FUNCTION "LAxisCtrl_UnpubReferencingVelocitySyncAxis" : LReal   // FC30638, SCL
TITLE = LAxisCtrl_UnpubReferencingVelocitySyncAxis
{ S7_Optimized_Access := 'TRUE' }
AUTHOR : tech.team.motioncontrol@siemens.com
FAMILY : AxisCtrl
VERSION : 1.1
// Support: tech.team.motioncontrol@siemens.com
   VAR_INPUT
      axis : TO_SynchronousAxis;   // Axis specification
   END_VAR
   // Ret_Val : axis.Homing.ReferencingVelocity
BEGIN
   // Read axis parameter
   #LAxisCtrl_UnpubReferencingVelocitySyncAxis := #axis.Homing.ReferencingVelocity;
END_FUNCTION

// ===== library: MasterCopy "LAxisCtrl_UnpubSensorTypePosAxis" =====

// folder: LAxisCtrl_Blocks/InternalSubBlocks/SensorType

FUNCTION "LAxisCtrl_UnpubSensorTypePosAxis" : DInt   // FC30643, SCL
TITLE = LAxisCtrl_UnpubSensorTypePosAxis
{ S7_Optimized_Access := 'TRUE' }
AUTHOR : tech.team.motioncontrol@siemens.com
FAMILY : AxisCtrl
VERSION : 1.1
// Support: tech.team.motioncontrol@siemens.com
   VAR_INPUT
      axis : TO_PositioningAxis;   // Axis specification
      index : Int;   // Index of sensor
   END_VAR
   // Ret_Val : axis.Sensor[index].Type
BEGIN
   // Read axis parameter
   #LAxisCtrl_UnpubSensorTypePosAxis := #axis.Sensor[#index].Type;
END_FUNCTION

// ===== library: MasterCopy "LAxisCtrl_UnpubSensorTypeSyncAxis" =====

// folder: LAxisCtrl_Blocks/InternalSubBlocks/SensorType

FUNCTION "LAxisCtrl_UnpubSensorTypeSyncAxis" : DInt   // FC30642, SCL
TITLE = LAxisCtrl_UnpubSensorTypeSyncAxis
{ S7_Optimized_Access := 'TRUE' }
AUTHOR : tech.team.motioncontrol@siemens.com
FAMILY : AxisCtrl
VERSION : 1.1
// Support: tech.team.motioncontrol@siemens.com
   VAR_INPUT
      axis : TO_SynchronousAxis;   // Axis specification
      index : Int;   // Index of sensor
   END_VAR
   // Ret_Val : axis.Sensor[index].Type
BEGIN
   // Read axis parameter
   #LAxisCtrl_UnpubSensorTypeSyncAxis := #axis.Sensor[#index].Type;
END_FUNCTION

// ===== library: MasterCopy "LAxisCtrl_typeGearOutCamOut" =====

// folder: LAxisCtrl_Types/LAxisCtrl_SubTypes

TYPE "LAxisCtrl_typeGearOutCamOut"
TITLE = LAxisCtrl_typeGearOutCamOut
// Support: tech.team.motioncontrol@siemens.com
   STRUCT
      slavePosition : LReal := 0.0;   // Stop position of following axis
      syncProfileReference : DInt := 1;   // Type of desynchronization (0: Desynchronize using dynamic behavior; 1: Desynchronize using leading value distance; 5: Cancel only a pending gearing / camming)
      masterStopDistance : LReal := 0.0;   // Leading value distance when "SyncProfileReference" = 1
      deceleration : LReal := -1.0;   // Deceleration for desynchronization (Value > 0.0: The specified value is used; Value = 0.0: Not permitted; Value < 0.0: Use of the default value configured in the technology object) when "SyncProfileReference" = 0
      jerk : LReal := -1.0;   // Jerk for desynchronization (Value > 0.0: Smooth velocity profile, the specified value is used; Value = 0.0: Trapezoidal velocity profile; Value < 0.0: Use of the default value configured in the technology object) when "SyncProfileReference" = 0
      syncOutDirection : DInt := 3;   // Desynchronization direction (1: Positive direction; 2: Negative direction; 3: Current direction)
      gearOutCamOutMode : DInt := -1;   // -1: Automatic detection whether to use a MC_GearOut or MC_CamOut; 0: Use of MC_GearOut; 1: Use of MC_CamOut
   END_STRUCT;
END_TYPE

// ===== library: MasterCopy "LAxisCtrl_typeGearInRelative" =====

// folder: LAxisCtrl_Types/LAxisCtrl_SubTypes

TYPE "LAxisCtrl_typeGearInRelative"
TITLE = LAxisCtrl_typeGearInRelative
// Support: tech.team.motioncontrol@siemens.com
   STRUCT
      ratioNumerator : DInt := 1;   // Gear ratio numerator (permitted integer values: -2147483648 to 2147483647; value 0 not permitted)
      ratioDenominator : DInt := 1;   // Gear ratio denominator (permitted integer values: 1 to 2147483647)
      acceleration : LReal := -1.0;   // Acceleration for synchronization (Value > 0.0: The specified value is used; Value = 0.0: Not permitted; Value < 0.0: Use of the default value configured in the technology object)
      deceleration : LReal := -1.0;   // Deceleration for synchronization (Value > 0.0: The specified value is used; Value = 0.0: Not permitted; Value < 0.0: Use of the default value configured in the technology object)
      jerk : LReal := -1.0;   // Jerk for synchronization (Value > 0.0: Smooth velocity profile, the specified value is used; Value = 0.0: Trapezoid velocity profile; Value < 0.0: Use of the default value configured in the technology object)
      ratioChangeOnTheFly : Bool := FALSE;   // TRUE: Changing gear ratio on-the-fly; FALSE: Ratio change requires a new rising edge at gearInRelative input
   END_STRUCT;
END_TYPE

// ===== library: MasterCopy "LAxisCtrl_Axis" =====

// folder: LAxisCtrl_Blocks

FUNCTION_BLOCK "LAxisCtrl_Axis"   // FB30616, SCL
TITLE = LAxisCtrl_Axis
{ S7_Optimized_Access := 'TRUE' }
AUTHOR : tech.team.motioncontrol@siemens.com
FAMILY : AxisCtrl
VERSION : 1.2
// Support: tech.team.motioncontrol@siemens.com
   VAR_INPUT
      enable : Bool := FALSE;   // TRUE: Enable functionality of FB
      enableAxis : Bool := FALSE;   // TRUE: Set axis enable; FALSE: Remove axis enable
      resetAxis : Bool := FALSE;   // Rising edge: Acknowledgment of technology alarms or restart of the axis (depending on configuration)
      openBrake : Bool := FALSE;   // TRUE: Unconditionally open holding brake if axis is not enabled (e.g. for service purposes)
      jogForward : Bool := FALSE;   // Rising edge: Move an axis in jog mode (forward); Falling edge: Stop jogging
      jogBackward : Bool := FALSE;   // Rising edge: Move an axis in jog mode (backward); Falling edge: Stop jogging
      moveVelocity : Bool := FALSE;   // Rising edge: Move an axis at constant velocity/speed
      stop : Bool := FALSE;   // Rising edge: Brake an axis until it comes to a standstill. Note: MC_Halt is triggered internally
      fastStop : Bool := FALSE;   // Rising edge: Brake an axis until it comes to a standstill (with fastStop dynamics). Note: MC_Halt is triggered internally
      torqueLimiting : Bool := FALSE;   // TRUE: Enable force/torque limiting
      homing : Bool := FALSE;   // Rising edge: Home axis
      posRelative : Bool := FALSE;   // Rising edge: Move an axis relative to its position when execution of the job began
      posAbsolute : Bool := FALSE;   // Rising edge: Move an axis to an absolute position
      posSuperimposed : Bool := FALSE;   // Rising edge: Start a superimposed positioning
      gearInRelative : Bool := FALSE;   // Rising edge: Start a gearing operation (relative)
      gearInAbsolute : Bool := FALSE;   // Rising edge: Start a gearing operation (absolute)
      gearOutCamOut : Bool := FALSE;   // Rising edge: End a gearing/camming operation
      camIn : Bool := FALSE;   // Rising edge: Start a camming operation
      phasing : Bool := FALSE;   // Rising edge: Start a phasing operation
      offset : Bool := FALSE;   // Rising edge: Start an offset operation
      axis : DB_ANY := 0;   // Reference to axis technology object to be controlled
      master : DB_ANY := 0;   // Reference to leading axis technology object for synchronous motion
      cam : DB_ANY := 0;   // Cam technology object
      configuration : "LAxisCtrl_typeAxisConfig";   // Structure for parameters
   END_VAR
   VAR_OUTPUT
      valid : Bool := FALSE;   // TRUE: Valid set of output values available at the FB
      busy : Bool := FALSE;   // TRUE: FB is working and new output values can be expected
      error : Bool := FALSE;   // TRUE: An error occurred while processing the FB
      status : Word := 16#7000;   // Current status of FB (16#0000 - 16#7FFF: Status of the FB, 16#8000 - 16#FFFF: Error identification)
      statusText : String[#STATUS_TEXT_LENGTH] := STRING#'STATUS_NO_CALL';   // Text of current status of FB
      subfunctionStatus : Word;   // Status of internally called subfunctions (ErrorID of Motion Control instructions)
      axisEnabled : Bool := FALSE;   // TRUE: The technology object is enabled. Motion commands can be executed
      resetActive : Bool := FALSE;   // TRUE: Reset/Restart of the axis is active
      commandBusy : Bool := FALSE;   // TRUE: The selected basic motion command is being executed
      commandDone : Bool := FALSE;   // TRUE: The selected basic motion command has completed without error
      commandAborted : Bool := FALSE;   // TRUE: The selected basic motion command has been aborted
      inVelocity : Bool := FALSE;   // TRUE: The setpoint velocity/speed was reached and will be maintained
      inLimitation : Bool := FALSE;   // TRUE: The drive is operating at the force/torque limit
      homingCommandBusy : Bool := FALSE;   // TRUE: Homing command is being executed
      homingCommandDone : Bool := FALSE;   // TRUE: Homing command has completed without error
      homingCommandAborted : Bool := FALSE;   // TRUE: Homing command has been aborted
      superimposedBusy : Bool := FALSE;   // TRUE: The selected superimposed motion command is being executed
      superimposedDone : Bool := FALSE;   // TRUE: The selected superimposed motion command has completed without error
      superimposedAborted : Bool := FALSE;   // TRUE: The selected superimposed motion command has been aborted
      superimposedStart : Bool := FALSE;   // TRUE: The selected superimposed motion is active
      inClamping : Bool := FALSE;   // TRUE: The drive is kept at the fixed stop (clamping), the axis position is within the positioning tolerance
      startSync : Bool := FALSE;   // TRUE: The axis is synchronizing to the leading axis / desynchronizing from the leading axis
      inSync : Bool := FALSE;   // TRUE: The axis is synchronized to the leading axis
      endOfProfile : Bool := FALSE;   // TRUE: The end of the cam has been reached. The output is displayed for at least one call when the cam is used cyclically
      inSimulation : Bool := FALSE;   // TRUE: Synchronous operation is being simulated
      jogSelected : Bool := FALSE;   // TRUE: Jogging is active
      moveVelocitySelected : Bool := FALSE;   // TRUE: Moving with constant velocity/speed is active
      stopSelected : Bool := FALSE;   // TRUE: Stopping is active
      fastStopSelected : Bool := FALSE;   // TRUE: Stopping is active (with fastStop dynamics)
      torqueLimitingSelected : Bool := FALSE;   // TRUE: Force/Torque limiting is active
      homingSelected : Bool := FALSE;   // TRUE: Homing is active
      posRelativeSelected : Bool := FALSE;   // TRUE: Relative positioning is active
      posAbsoluteSelected : Bool := FALSE;   // TRUE: Absolute positioning is active
      posSuperimposedSelected : Bool := FALSE;   // TRUE: Superimposed positioning is active (See also outputs: superimposedBusy, superimposedDone, superimposedAborted)
      gearInRelativeSelected : Bool := FALSE;   // TRUE: Relative gearing is active (See also outputs: commandBusy, commandDone, commandAborted, inSync)
      gearInAbsoluteSelected : Bool := FALSE;   // TRUE: Absolute gearing is active (See also outputs: commandBusy, commandDone, commandAborted, startSync, inSync)
      gearOutCamOutSelected : Bool := FALSE;   // TRUE: End a gearing/camming operation is active (See also outputs: commandBusy, commandDone, commandAborted, startSync)
      camInSelected : Bool := FALSE;   // TRUE: Camming is active (See also outputs: commandBusy, commandDone, commandAborted, startSync, inSync)
      phasingSelected : Bool := FALSE;   // TRUE: Phasing is active (See also outputs: superimposedBusy, superimposedDone, superimposedAborted, superimposedStart)
      offsetSelected : Bool := FALSE;   // TRUE: Offset is active (See also outputs: superimposedBusy, superimposedDone, superimposedAborted, superimposedStart)
      diagnostics : "LAxisCtrl_typeDiagnostics";   // Diagnostics structure
   END_VAR
   VAR
      statStatusOld : Word;   // Old value of statStatus
      statStatusText : String[#STATUS_TEXT_LENGTH] := STRING#'STATUS_NO_CALL';   // Internal text of current status of FB
      statErrorUserCleared : Bool := FALSE;   // Error occurred that can only be solved by user; rising edge at enable input necessary
      statErrorAutoCleared : Bool := FALSE;   // Error occurred that can be acknowledged by FB
      statStatus : Word := 16#7000;   // Internal variable for status
      statSubfunctionStatus : Word := 16#0000;   // Internal variable for subfunction status
      statDiagnostics : "LAxisCtrl_typeDiagnostics";   // Internal variable for diagnostics
      statEnableOld : Bool := FALSE;   // Old value of enable for edge detection
      statFBState : SInt := 1;   // State of FB (function block state machine)
      statFirstCycleReset : Bool := TRUE;   // TRUE: First cycle of reset command
      statPowerErrorOld : Bool := FALSE;   // Old value of LAnyAxis_MC_Power.error
      statResetState : Int := 0;   // State of reset command
      statFirstCycleResetError : Bool := FALSE;   // TRUE: First cycle of error in reset command
      statExtendedCommand : DWord := 16#0000_0000;   // Variable for requested extended command (e.g. resetAxis, torquelimiting, homing)
      statExtendedCommandOld : DWord := 16#0000_0000;   // Old value of variable for requested extended command
      statEnableAxisOld : Bool := FALSE;   // Old value of enableAxis for edge detection
      statEmptyDiagnostics : "LAxisCtrl_typeDiagnostics";   // Internal empty diagnostic structure
      statHomingOld : Bool := FALSE;   // Old value of variable for homing command input
      statFirstCycleHoming : Bool := TRUE;   // TRUE: First cycle in homing command
      statPassiveHomingState : DInt := -10;   // Current selected passive homing mode
      statExeOfHoming : Int := 1;   // Current state of execution of homing command
      statBasicCommand : DWord := 16#0000_0000;   // Variable for requested basic motion command
      statBasicCommandOld : DWord := 16#0000_0000;   // Old value of variable for requested basic motion command
      statBasicMotionState : DInt := 0;   // State of selected basic motion command
      statExeOfBasicMotion : Int := 1;   // State of execution of current state of basic motion
      statFirstCycleBasicMotion : Bool := TRUE;   // TRUE: First cycle in respective state fo basic motion functionality
      statApplicativeBasicMotionError : Bool := FALSE;   // TRUE: applicative error occurred (e.g. invalid direction configured)
      statVelocityChangeOnTheFly : Bool := FALSE;   // Velocity change on the fly is active
      statBasicVelocity : LReal := 0.0;   // Internal variable for velocity
      statBasicAcceleration : LReal := 0.0;   // Internal variable for acceleration
      statBasicAbortAcceleration : Bool := FALSE;   // FALSE: The current acceleration at the start of the job is reduced using the configured jerk. Afterwards, the deceleration builds up; TRUE: The acceleration is set to 0.0 at the start of the job, and the deceleration immediately builds up.
      statBasicDeceleration : LReal := 0.0;   // Internal variable for deceleration
      statBasicJerk : LReal := 0.0;   // Internal variable for jerk
      statPositionControlled : Bool := TRUE;   // FALSE: Non position-controlled operation; TRUE: Position-controlled operation
      statFirstCycleDone : Bool := FALSE;   // TRUE: First cycle of done at fastStop
      statTorqueLimitingState : SInt := 0;   // Current executed state for torquelimiting functionality
      statTorqueLimitingErrorOld : Bool := FALSE;   // TRUE: Error at Torquelimiting occurred last cycle
      statTorqueLimit : LReal := -1.0;   // Value of force/torque limiting (in the configured unit of measurement)
      statJogMode : DInt := 0;   // Current selected jog mode
      statDirection : Int := 0;   // Internal variable for direction of rotation of the axis
      statStopWithoutSignalization : Bool;   // Internal variable for stopOnError function
      statBrakeOpened : Bool;   // Brake is openend
      statBrakeChangeActive : Bool;   // Brake change active
      statOpenBrakeOld : Bool;   // Edge detection
      statSupImpVelocity : LReal := 0.0;   // Internal variable for velocity
      statSupImpAcceleration : LReal := 0.0;   // Internal variable for acceleration
      statSupImpDeceleration : LReal := 0.0;   // Internal variable for deceleration
      statSupImpJerk : LReal := 0.0;   // Internal variable for jerk
      statHomingPosition : LReal := 0.0;   // The specified value is used according to the selected "Mode".
      statHomingSubState : SInt := 0;   // Current subState of execution of homing functionality
      statIncJogSubState : SInt := 0;   // Current subState of execution of jog incremental functionality
      statIncJogStartPosition : LReal := 0.0;   // Last stored axis position (for incremental jogging)
      statIncJogDirectionOld : Int := 0;   // Old value of direction of executing incremental jogging
      statIncrement : LReal := 0.0;   // Jog Incremental: distance of Increment (positive or negative)
      statIncJogDistance : LReal := 0.0;   // Jog Incremental: current distance to destination position
      statResetIncJog : Bool := TRUE;   // TRUE: First cycle in incremental jogging state (detection of new increment)
      statPosition : LReal := 0.0;   // Internal variable for position
      statPositionChangeOnTheFly : Bool := FALSE;   // Position change on the fly is active
      statHomingMode : Int := 0;   // Operating Mode of LAnyAxis_MC_HOME command
      statActiveHomingState : DInt := -10;   // Current selected active homing mode
      statSupImpCommand : DWord := 16#0000_0000;   // Variable for requested superimposed motion command
      statSupImpCommandOld : DWord := 16#0000_0000;   // Old value of variable for requested superimposed motion command
      statSupImpMotionState : DInt := 0;   // Current selected superimposed motion functionality
      statExeOfSupImpMotionState : Int := 1;   // Current state of execution of superimposed basic motion
      statFirstCycleSupImpMotion : Bool := TRUE;   // TRUE: First cycle in positioning (superimposed) functionality
      statSupImpMotionPosition : LReal := 0.0;   // Position setpoint (for posSuperimposed command)
      statApplicativeSupImpMotionError : Bool := FALSE;   // TRUE: applicative error occurred (e.g. invalid direction configured)
      statRatioChangeOnTheFly : Bool := FALSE;   // Ratio change on the fly is active
      statRatioNumerator : DInt := 1;   // Gear ratio numerator
      statRatioDenominator : DInt := 1;   // Gear ratio denominator
      statChangePhaseShiftOnTheFly : Bool := FALSE;   // Phase shift change on the fly is active
      statChangeOffsetOnTheFly : Bool := FALSE;   // Offset change on the fly is active
      statPhaseShift : LReal := 0.0;   // Relative/Absolute master value shift
      statPhaseAbsolute : Bool := TRUE;   // Indicates the type of phase shift (TRUE: The phase shift is taken over as an absolute value; FALSE: The phase shift is added to an existing offset)
      statOffsetAbsolute : Bool := FALSE;   // Indicates the type of offset shift (TRUE: The offset shift is taken over as an absolute value; FALSE: The offset shift is added to an existing offset)
      statOffsetValue : LReal := 0.0;   // Relative/Absolute offset
      statTypeAxis : Int;   // Type of axis
      statSupImpProfileReference : DInt := 0;   // Internal variable
      statSupImpDistance : LReal := 0.0;   // Internal variable
      statSupImpStartPosition : LReal := 0.0;   // Internal variable
      statSupImpDirection : DInt := 0;   // Internal variable
      statEnableAxis : Bool := FALSE;   // Internal variable for enabling axis
      statSyncMotionSimulationState : SInt := 0;   // Current executed state for synchronized motion simulation
      statSynchronizedMotionErrorOld : Bool := FALSE;   // Old value of LAnyAxis_MC_SynchronizedMotionSimulation.error
      statMainSelectionState : Int := 0;   // Current executed State for execution of basic motion commands or reset of waiting gearing / camming commands
      statMasterSyncPosition : LReal := 0.0;   // Synchronous position of leading axis. Position of the following axis starting from which the leading and following axes move synchronously
      statSlaveSyncPosition : LReal := 0.0;   // Synchronous position of leading axis. Position of the leading axis starting from which the leading and following axes move synchronously
      statBasicSyncDirection : DInt := 1;   // Direction of synchronization
      statBasicMasterStartDistance : LReal := 0.0;   // Master value distance (when "SyncProfileReference" = 1)
      statBasicSyncProfileReference : DInt := 0;   // Type of synchronization
      statApplicationMode : DInt := 0;   // Application of cam
      statCam : DB_ANY := 0;   // Internal variable for cam
      statWaitingFunctionState : DInt := 0;   // Internal variable for waiting function state
      statWaitingFunctionStateAbortAutomatic : DInt := -1;   // Internal variable for waiting function state
      statFunctionState : DInt := 0;   // Internal variable for function state
      statGearAndCamOutMode : DInt := 0;   // Internal variable
      statSyncOutState : DInt;   // Internal variable
      statAxis : DB_ANY;   // Internal axis reference
      instPower : "LAnyAxis_MC_Power";   // Instance of LAnyAxis_MC_Power
      instReset : "LAnyAxis_MC_Reset";   // Instance of LAnyAxis_MC_Reset
      instHome : "LAnyAxis_MC_Home";   // Instance of LAnyAxis_MC_Home
      instHalt : "LAnyAxis_MC_Halt";   // Instance of LAnyAxis_MC_Halt
      instMoveJog : "LAnyAxis_MC_MoveJog";   // Instance of LAnyAxis_MC_MoveJog
      instTorqueLimiting : "LAnyAxis_MC_TorqueLimiting";   // Instance of LAnyAxis_MC_TorqueLimiting
      instMoveVelocity : "LAnyAxis_MC_MoveVelocity";   // Instance of LAnyAxis_MC_MoveVelocity
      instSetAxisSTW : "LAnyAxis_MC_SetAxisSTW";   // Instance of LAnyAxis_MC_SetAxisSTW
      instMoveRelative : "LAnyAxis_MC_MoveRelative";   // Instance of LAnyAxis_MC_MoveRelative
      instMoveAbsolute : "LAnyAxis_MC_MoveAbsolute";   // Instance of LAnyAxis_MC_MoveAbsolute
      instMoveSuperimposed : "LAnyAxis_MC_MoveSuperimposed";   // Instance of LAnyAxis_MC_MoveSuperimposed
      instGearIn : "LAnyAxis_MC_GearIn";   // Instance of LAnyAxis_MC_GearIn
      instPhasingAbsolute : "LAnyAxis_MC_PhasingAbsolute";   // Instance of LAnyAxis_MC_PhasingAbsolute
      instPhasingRelative : "LAnyAxis_MC_PhasingRelative";   // Instance of LAnyAxis_MC_PhasingRelative
      instOffsetAbsolute : "LAnyAxis_MC_OffsetAbsolute";   // Instance of LAnyAxis_MC_OffsetAbsolute
      instOffsetRelative : "LAnyAxis_MC_OffsetRelative";   // Instance of LAnyAxis_MC_OffsetRelative
      instGearInPos : "LAnyAxis_MC_GearInPos";   // Instance of LAnyAxis_MC_GearInPos
      instGearOut : "LAnyAxis_MC_GearOut";   // Instance of LAnyAxis_MC_GearOut
      instCamIn : "LAnyAxis_MC_CamIn";   // Instance of MC_CamIn
      instCamOut : "LAnyAxis_MC_CamOut";   // Instance of LAnyAxis_MC_CamOut
      instSyncMotionSimulation : "LAnyAxis_MC_SynchronizedMotionSimulation";   // Instance of LAnyAxis_MC_SynchronizedMotionSimulation
   END_VAR
   VAR_TEMP
      tempEnable : Bool;   // Temporary variable for enable FB
      tempNewExtendedCmd : DInt;   // Temporary variable for extended command
      tempEnableAxis : Bool;   // Temporary variable for enableAxis
      tempErrorInCmd : Bool;   // Temporary variable for error in actual command
      tempRisingCmd : DWord;   // Temporary DWord which indicates all rising edges of command word
      tempStopCmdSelected : Bool;   // TRUE: Stop or faststop selected in current cycle
      tempOpenBrake : Bool;   // Temporary variable for open brake
      tempDword : DWord;   // Temporary DWord for evaluation of rising edges of basic command word
      tempIndex : Int;   // Temporary index
      tempCountRisEdges : USInt;   // Temporary counter for rising edges in command word
      tempNewBasicMotionCmd : DInt;   // Temporary variable for basic motion command
      tempStateChangeActive : Bool;   // TRUE: State change is active, stay in loop for one more cycle
      tempStatusWord : DWord;   // Temporary variable for statusword of axis
      tempNewSupImpCmd : DInt;   // Temporary variable for superimposed motion command
      tempHoming : Bool;   // Temporary variable for homing command
   END_VAR
   VAR CONSTANT
      EXTERNAL_ENCODER : Int := 1;   // Axis type: External encoder
      SPEED_AXIS : Int := 2;   // Axis type: Speed axis
      POS_AXIS : Int := 3;   // Axis type: Positioning axis
      SYNC_AXIS : Int := 4;   // Axis type: Synchronous axis
      STATUS_TEXT_LENGTH : Int := 39;   // Length of status text
      AXIS_MOTION : SInt := 1;   // State of FB: MotionState, new commands are evaluated
      FB_ERROR : SInt := 5;   // State of FB: Error, falling edge at FB_ENABLE required
      CMD_NO_SELECTION : DWord := 16#0000_0000;   // No command is selected
      NO_SELECTION : Int := 0;   // State of basicMotion/superimposedMotion: No execution of a command
      AXIS_FAST_STOPPING : SInt := 2;   // State of FB: StoppingState, MC_HALT is executed, new commands are not evaluated
      AXIS_STOP_ON_ERROR_SELECTION : SInt := 3;   // State of FB: ErrorState: Selection if StopOnError must be executed (depending on configuration)
      AXIS_STOP_ON_ERROR_EXECUTION : SInt := 4;   // State of FB: ErrorState: Execution of StopOnError
      FAST_STOP_SELECTED : Int := 1;   // State of basicMotion: Execution of fast stop command
      STOP_SELECTED : Int := 2;   // State of basicMotion: Execution of stop command
      JOG_FORWARD_SELECTED : Int := 4;   // State of basicMotion: Execution of jog forward command
      JOG_BACKWARD_SELECTED : Int := 8;   // State of basicMotion: Execution of jog backward command
      JOG_FW_AND_BW_SELECTED : Int := 12;   // State of basicMotion: Execution of jog command if forward and backward are selected
      MOVE_VELOCITY_SELECTED : Int := 16;   // State of basicMotion: Execution of move velocity command
      ACTIVE_HOMING_SELECTED : Int := 1024;   // State of basicMotion: Execution of active homing command
      POS_RELATIVE_SELECTED : Int := 32;   // State of basicMotion: Execution of position command (relative)
      POS_ABSOLUTE_SELECTED : Int := 64;   // State of basicMotion: Execution of position command (absolute)
      GEAR_IN_RELATIVE_SELECTED : Int := 128;   // State of basicMotion: Execution of gearIn command
      GEAR_IN_ABSOLUTE_SELECTED : Int := 256;   // State of basicMotion: Execution of gearInPos command
      CAM_IN_SELECTED : Int := 512;   // State of basicMotion: Execution of camIn command
      GEAR_OUT_CAM_OUT_SELECTED : Int := 2048;   // State of basicMotion: Execution of gear and camOut command
      POS_SUPERIMPOSED_SELECTED : Int := 1;   // State of superimposedMotion: Execution of posSuperimposed command
      PHASING_SELECTED : Int := 2;   // State of superimposedMotion: Execution of phasing command
      OFFSET_SELECTED : Int := 4;   // State of superimposedMotion: Execution of offset command
      CMD_IDLE : Int := 0;   // State of basicMotion command: No execution
      CMD_BUSY : Int := 1;   // State of basicMotion command: Subsequent call
      CMD_DONE : Int := 2;   // State of basicMotion command: Finished with "DONE"
      CMD_ABORTED : Int := 4;   // State of basicMotion command: Finished with "ABORTED"
      CMD_ERROR : Int := 8;   // State of basicMotion command: Finished with "ERROR"
      CMD_END_PROCESS : Int := 16;   // State of basicMotion command: Finished with other reason
      JOG_MODE_CONTINUOUS : Int := 0;   // Jogmode continuous selected (MC_MOVEJOG)
      NO_TORQUE_LIMITING_ACTIVE : SInt := 0;   // State of torquelimiting command: Not enabled
      TORQUE_LIMTING_SELECTED : SInt := 1;   // State of torquelimiting command: Torquelimiting is active
      TORQUE_LIMITING_DISABLE : SInt := 10;   // State of torquelimiting command: Torquelimiting is disabling
      BITPOSITION_BASIC_MOTION_CMD : SInt := 4;   // First bitposition for detecting rising edges at basic motion command word
      BIT_POS_LAST : SInt := 15;   // Last bitposition for detecting rising edges at command word
      SPECIFIED_DIR : Int := 0;   // The sign of the velocity specified at the "Velocity" parameter defines the direction of rotation.
      MASK_STW_BIT12 : Word := 16#1000;   // Bit 12 in STW
      NO_HOMING_ACTIVE : SInt := -10;   // State of homing command: No homing active
      STANDARD_HOMING : SInt := -1;   // State of homing command: (Standard) homing with MC_HOME
      BITPOSITION_SUPERIMPOSED_MOTION_CMD : SInt := 0;   // First bitposition for detecting rising edges at superimposed motion command word
      FIXED_STOP_DETECTION_ACTIVE : SInt := 2;   // State of torquelimiting command: Homing on fixed stop is active
      FIXED_STOP_DETECTION_FINISHED : SInt := 3;   // State of torquelimiting command: Homing on fixed stop is finished
      FIXED_STOP_DETECTION_ERROR_IN_CLAMPING : SInt := 5;   // State of torquelimiting command: Error occurred at homing on fixed stop process, axis is in clamping
      FIXED_STOP_DETECTION_ERROR_NOT_IN_CLAMPING : SInt := 6;   // State of torquelimiting command: Error occurred at homing on fixed stop process, axis is not in clamping
      HOMING_ON_FIXED_STOP : SInt := 0;   // State of homing command: Applicative homing on fixed stop process active
      HOMING_ON_FIXED_STOP_WITH_MOVING_OUT_OF_CLAMPING : SInt := 1;   // State of homing command: Applicative homing on fixed stop with moving out of clamping process active.
      HOMING_ON_FIXED_STOP_WITH_MOVING_TO_TARGET_POSITION : SInt := 2;   // State of homing command: Applicative homing on fixed stop with moving to target position process active.
      DISTANCE_SCALING : LReal := 1.05;   // Scaling factor for moving out of clamping. 1.0 = positioning window
      MODE_FIXED_STOP_DETECTION : Int := 1;   // Fixed stop detection (Mode for MC_TORQUELIMITING)
      FORWARD_DIR : Int := 1;   // Positive/Forward direction of rotation
      BACKWARD_DIR : Int := 2;   // Negative/Backward direction of rotation
      SHORTEST_WAY_DIR : Int := 3;   // Shortest path
      DIRECT_HOMING : Int := 0;   // Direct homing (absolute). Parameter "position" at MC_HOME is effective
      ACTIVE_HOMING : Int := 3;   // Active homing. Parameter "position" at MC_HOME is effective
      ACTIVE_HOMING_TO_DEF_VALUE : Int := 5;   // Active homing. The configured home position value in technology object is effective
      ABSOLUTE_ENCODER_ADJUSTMENT : Int := 7;   // Absolute encoder adjustment (absolute)
      INCREMENTAL_ENCODER : Int := 0;   // Encodertype INCREMENTAL
      HOMING_IDLE : SInt := 0;   // SubState of homing on fixed stop process: Idle
      HOMING_FIXED_STOP_DETECTION : SInt := 1;   // SubState of homing on fixed stop process: Detecting fixed stop
      HOMING_PROCESS : SInt := 2;   // SubState of homing on fixed stop process: Homeprocess (MC_HOME)
      HOMING_POSITION : SInt := 3;   // SubState of homing on fixed stop process: Positioning to homeposition
      INC_JOG_IDLE : SInt := 0;   // Substate of incremental jog process: Idle
      INC_JOG_START : SInt := 1;   // Substate of incremental jog process: Start moving
      INC_JOG_STOP : SInt := 3;   // Substate of incremental jog process: Stop moving
      JOG_MODE_NEW_INCREMENT : Int := 1;   // Jogmode incremental selected - start always with new increment when command is selected
      JOG_MODE_CONTINUE_INCREMENT : Int := 2;   // Jogmode incremental selected - continue with increment when command is selected again
      APPLICATION_MODE_ONCE : Int := 0;   // Application of the cam: Once/not cyclic (MC_CAMIN)
      CALL_BASIC_MOTION : Int := 0;   // State of MainSelectionState: Regular execution of basic motion commands
      ABORT_WAITING_GEARINPOS_OR_CAMIN : Int := 1;   // State of MainSelectionState: Reset of waiting synchronous commands
      AXIS_NOT_IN_SIM : SInt := 0;   // State of motionSimulation: Axis is not in simulation
      AXIS_STATE_SET_SIM : SInt := 1;   // State of motionSimulation: Setting axis in simulation
      AXIS_DISABLE : SInt := 2;   // State of motionSimulation: Disable axis
      AXIS_STATE_IN_SIM : SInt := 3;   // State of motionSimulation: Axis is in simulation
      AXIS_ENABLE : SInt := 4;   // State of motionSimulation: Enable axis
      AXIS_STATE_RESET_SIM : SInt := 5;   // State of motionSimulation: Resetting axis simulation
      CANCEL_ONLY_WAITING_GEARING_CAMMING : DInt := 5;   // Mode for MC_GearOut / MC_CamOut instruction
      WFS_FS_NO_OPERATION : DInt;   // No operation active or waiting
      WFS_FS_GEARIN : DInt := 1;   // Function state / Waiting function state: GearIn
      WFS_FS_GEARINPOS : DInt := 2;   // Function state / Waiting function state: GearInPos
      WFS_FS_CAMIN : DInt := 3;   // Function state / Waiting function state: CamIn
      WFS_FS_GEAROUT : DInt := 4;   // Function state / Waiting function state: Gearout
      WFS_FS_CAMOUT : DInt := 5;   // Function state / Waiting function state: CamOut
      SYNCOUT_MODE_AUTOMATIC : DInt := -1;   // GearOutCamOut mode: Automatic
      SYNCOUT_MODE_GEAROUT : DInt := 0;   // GearOutCamOut mode: GearOut
      SYNCOUT_MODE_CAMOUT : DInt := 1;   // GearOutCamOut mode: CamOut
      SYNCOUT_STATE_CHECK_WAITING : Int := 1;   // Sync out state
      SYNCOUT_STATE_GEAROUT_WAITING_BUSY : Int := 2;   // Sync out state
      SYNCOUT_STATE_CAMOUT_WAITING_BUSY : Int := 3;   // Sync out state
      SYNCOUT_STATE_CHECK_ACTIVE : Int := 4;   // Sync out state
      SYNCOUT_STATE_GEAROUT_ACTIVE_BUSY : Int := 5;   // Sync out state
      SYNCOUT_STATE_CAMOUT_ACTIVE_BUSY : Int := 6;   // Sync out state
      SYNCOUT_STATE_DONE : Int := 7;   // Sync out state
      SYNCOUT_STATE_ABORTED : Int := 8;   // Sync out state
      SYNCOUT_STATE_ERROR : Int := 9;   // Sync out state
      STATUS_NO_CALL : Word := 16#7000;   // No call of FB
      STATUS_FB_FIRST_CALL : Word := 16#7001;   // First cycle of FB after enabling
      STATUS_SUBSEQUENT_CALL : Word := 16#7002;   // FB enabled
      ERR_INVALID_BASIC_MOTION_CMD : Word := 16#8001;   // Invalid basic command selected (rising edge at 2 or more basic motion command inputs)
      ERR_INVALID_EXTENDED_CMD : Word := 16#8002;   // Invalid extended command selected (rising edge at torque limiting and homing on fixed stop)
      ERR_INVALID_SUPERIMPOSED_MOTION_CMD : Word := 16#8003;   // Invalid superimposed command selected (rising edge at 2 or more superimposed motion command inputs)
      ERR_INVALID_GEAROUT_CAMOUT_MODE : Word := 16#820D;   // Error invalid mode for gearOutCamOut instruction
      ERR_INVALID_SYNCHRONIZED_EXTENDED_MODE : Word := 16#820E;   // Error invalid extended mode for synchronized motion simulation functionality
      ERR_INVALID_JOG_MODE : Word := 16#8201;   // Invalid jog mode selected
      ERR_INVALID_HOMING_EXTENDED_MODE : Word := 16#8202;   // Command Error: Invalid extended homing mode selected
      ERR_TORQUE_LIMITING_NOT_ALLOWED : Word := 16#8203;   // Error during extended homing command - torque limiting not allowed during homing on fixed stop is active or axis in clamping
      ERR_INVALID_JOG_DIR : Word := 16#8204;   // Invalid direction selected (jog forward and jog backward)
      ERR_INVALID_POS_RELATIVE_DIR : Word := 16#8205;   // Invalid direction is set for relative positioning command
      ERR_INVALID_POS_SUPERIMPOSED_DIR : Word := 16#8206;   // Invalid direction is set for superimposed positioning command
      ERR_HOMING_MODE_NOT_ALLOWED : Word := 16#8207;   // Passive/Direct homing is not allowed during extended homing mode (homing on fixed stop process) is active
      ERR_MODULO_NOT_ALLOWED : Word := 16#8208;   // Extended homing mode (homing on fixed stop process) is not allowed with modulo axis
      ERR_INVALID_TORQUE_LIMIT : Word := 16#8209;   // Configured torque limit value for extended homing mode (homing on fixed stop process) = 0
      ERR_INVALID_VELOCITY : Word := 16#820A;   // Configured velocity (in technology object) for active homing = 0
      ERR_INVALID_AXIS : Word := 16#820B;   // Illegal specification of the technology object
      ERR_INVALID_TARGET_POSITION : Word := 16#820C;   // Invalid target position configured for extended homing mode
      ERR_MC_POWER : Word := 16#8600;   // Error occurred during MC_POWER command
      ERR_MC_RESET : Word := 16#8601;   // Error occurred during MC_RESET command
      ERR_MC_HOME : Word := 16#8602;   // Error occurred during MC_HOME command
      ERR_MC_TORQUELIMITING : Word := 16#8603;   // Error occurred during MC_TORQUELIMITING command
      ERR_MC_HALT : Word := 16#8604;   // Error occurred during MC_HALT command
      ERR_MC_MOVEJOG : Word := 16#8605;   // Error occurred during MC_MOVEJOG command (continuous jogging)
      ERR_MC_MOVEVELOCITY : Word := 16#8606;   // Error occurred during MC_MOVEVELOCITY command
      ERR_MC_MOVERELATIVE : Word := 16#8607;   // Error occurred during MC_MOVERELATIVE command
      ERR_MC_MOVEABSOLUTE : Word := 16#8608;   // Error occurred during MC_MOVEABSOLUTE command
      ERR_MC_MOVESUPERIMPOSED : Word := 16#8609;   // Error occurred during MC_MOVESUPERIMPOSED command
      ERR_MC_GEARIN : Word := 16#860A;   // Error occurred during MC_GEARIN command
      ERR_MC_PHASINGABSOLUTE : Word := 16#860B;   // Error occurred during MC_PHASINGABSOLUTE command
      ERR_MC_PHASINGRELATIVE : Word := 16#860C;   // Error occurred during MC_PHASINGRELATIVE command
      ERR_MC_CAMIN : Word := 16#860D;   // Error occurred during MC_CAMIN command
      ERR_MC_GEARINPOS : Word := 16#860E;   // Error occurred during MC_GEARINPOS command
      ERR_MC_SYNCHRONIZEDMOTIONSIMULATION : Word := 16#860F;   // Error occurred during MC_SYNCHRONIZEDMOTIONSIMULATION command
      ERR_MC_OFFSETABSOLUTE : Word := 16#8610;   // Error occurred during MC_OFFSETABSOLUTE command
      ERR_MC_OFFSETRELATIVE : Word := 16#8611;   // Error occurred during MC_OFFSETRELATIVE command
      ERR_MC_CAMOUT : Word := 16#8612;   // Error occurred during MC_CAMOUT command
      ERR_MC_GEAROUT : Word := 16#8613;   // Error occurred during MC_GEAROUT command
      ERR_UNDEFINED_FB_STATE : Word := 16#8700;   // Error due to an undefined FB state
      ERR_UNDEFINED_RESET_STATE : Word := 16#8701;   // Error due to an undefined reset state
      ERR_UNDEFINED_BASIC_MOTION_STATE : Word := 16#8702;   // Error due to an undefined basic motion state
      ERR_UNDEFINED_TORQUE_LIMITING_STATE : Word := 16#8703;   // Error due to an undefined torque limiting state
      ERR_UNDEFINED_INCREMENTAL_JOG_STATE : Word := 16#8704;   // Error due to an undefined incremental jog state
      ERR_UNDEFINED_INCREMENTAL_JOG_SUBSTATE : Word := 16#8705;   // Error due to an undefined incremental jog substate
      ERR_UNDEFINED_EXTENDED_HOMING_STATE : Word := 16#8706;   // Error due to an undefined homing state
      ERR_UNDEFINED_EXTENDED_HOMING_SUBSTATE : Word := 16#8707;   // Error due to an undefined homing substate
      ERR_UNDEFINED_SUPERIMPOSED_MOTION_STATE : Word := 16#8708;   // Error due to an undefined superimposed motion state
      ERR_UNDEFINED_MOTION_SIMULATION_STATE : Word := 16#8709;   // Error due to an undefined synchronized motion simulation state
      ERR_UNDEFINED_MAIN_SELECTION_STATE : Word := 16#870A;   // Error due to an undefined main selection state
   END_VAR
BEGIN
   REGION HEADER
     //================================================================================
     // SIEMENS AG
     // (c)Copyright 2021 All Rights Reserved
     //--------------------------------------------------------------------------------
     // Library: LAxisCtrl 
     // Tested with: S7-1515T-2 PN
     // Engineering: TIA Portal V17
     // Restrictions: -
     // Requirements: S7-1500/S7-1500T FW 2.9
     //               LAnyAxis V1.1                                                                                         
     // Functionality: This function block offers basic functionalities for axis control
     // Support: tech.team.motioncontrol@siemens.com
     // Note: Parameter comments are only available in language 'English (United States)'
     //--------------------------------------------------------------------------------
     // Change log table:
     // Version  Date        Expert in charge  Changes applied
     // 01.00.01 12.10.2016  RS                First released version
     // 01.00.02 29.03.2017  RS                Added support information
     //                                        TorqueLimiting at FB Enable                                                   
     //                                        Block is compilable with V14 SP1
     //                                        Output 'done' is set at endOfProfile of CamIn command (applicationMode ONCE)  
     //                                        fastStop: Use TO emergency stop deceleration in case of configured value <= 0 
     //                                        fastStop: Configured jerk value is always used                                
     // 01.00.03 14.06.2017  RS                Reset MC_TORQUELIMITING instance with disable of FB                           
     //                                        Bugfix of error handling for MC_TORQUELIMITING                                
     //                                        Homing on fixed stop: Use always torque value in homing configuration         
     // 01.00.04 14.12.2017  RS                Initialize diagnostics at rising edge of torquelimiting command               
     //                                        Check of cam (with TYPEOFDB) at start of camIn command                        
     // 01.00.05 30.09.2019  RS                Bugfixes
     //                                        Dont abort waiting sync commands if new gearinAbsolute or camIn or gearIn commands are set   
     //                                        Ratio on the fly: use also new dynamics if "on the fly value" changed         
     //                                        Stop on Error function: No error display if error at MC_Halt                  
     //                                        New extended homing mode: 1: Homing on fixed stop with moving out of clamping                        
     // 01.01.00 31.03.2020  RS                New output "subfunctionStatus"
     //                                        Change of parameter configuration: INOUT --> IN
     //                                        New input: "open brake"                                                       
     //                                        Optimized function: "abort waiting gearing commands"                          
     //                                        Stop on Error function: Error and status outputs remain also if internally        
     //                                        called MC_Halt instruction is executed                                        
     //                                        Output "diagnostics" is only written at end of block                          
     // 01.02.00 26.04.2021  RS                New output "statusText"
     //                                        New extended homing mode: 2: Homing on fixed stop with moving to target position   
     //                                        New feature: Automatic enabling of synchronized motion simulation when axis gets disabled  
     //                                        Update Motion Control V6.0 (MC_Offset_XXX, MC_Phasing_XXX, MC_GearOut; MC_CamOut)         
     //                                        FastStop command aborts waiting synchronous operations                        
     //                                        Bugfix synchronized motion simulation
     // 01.02.01 01.10.2021  RS                Bugfix synchronized motion simulation ('syncMotionSimulationExtendedMode' = -1):
     //                                        Axis is disabled (powered off) now, when parameter 'syncMotionSimulation' is set
     //                                        and no synchronous operation is active (<TO>.StatusWord.X22 = TRUE)
     //================================================================================
   END_REGION

   //----------------------------------------------------------------------------------------------
   // Enable / disable FB
   //----------------------------------------------------------------------------------------------
   REGION ENABLE_FB
     #tempEnable := #enable; // Create temporary process image
     IF NOT #tempEnable AND #statEnableOld THEN
       REGION FALLING_EDGE_AT_ENABLE_FB

         // Reset outputs 
         // ==========================================================
         // Error and valid outputs are reset with falling edge of enable input
         #error := FALSE;
         #valid := FALSE;
         #status := #STATUS_NO_CALL;
         #statusText := STRING#'STATUS_NO_CALL';
         #subfunctionStatus := #statSubfunctionStatus := 16#0; // V1.1.0

         // Reset status outputs
         #axisEnabled := FALSE;
         #resetActive := FALSE;

         // Reset outputs for homing commands
         #homingCommandBusy := FALSE;
         #homingCommandDone := FALSE;
         #homingCommandAborted := FALSE;
         #homingSelected := FALSE;
         // Reset outputs for torquelimiting command
         #torqueLimitingSelected := FALSE;
         #inLimitation := FALSE;

         // Reset outputs for basic motion commands
         #commandDone := FALSE;
         #commandBusy := FALSE;
         #commandAborted := FALSE;
         #inVelocity := FALSE;
         #fastStopSelected := FALSE;
         #stopSelected := FALSE;
         #jogSelected := FALSE;
         #moveVelocitySelected := FALSE;
         // Outputs for for up to LAxisCtrl_PosAxis
         #posRelativeSelected := FALSE;
         #posAbsoluteSelected := FALSE;
         #inClamping := FALSE;

         // Reset outputs for superimposed motion commands
         #superimposedBusy := FALSE;
         #superimposedDone := FALSE;
         #superimposedAborted := FALSE;
         #superimposedStart := FALSE;
         #posSuperimposedSelected := FALSE;
         #startSync := FALSE;
         #inSync := FALSE;
         #endOfProfile := FALSE;
         #gearInRelativeSelected := FALSE;
         #inSimulation := FALSE;
         #gearInAbsoluteSelected := FALSE;
         #phasingSelected := FALSE;
         #offsetSelected := FALSE;
         #camInSelected := FALSE;
         #gearOutCamOutSelected := FALSE;

         // Reset internal variables
         // ==========================================================
         #statErrorUserCleared := FALSE;
         #statErrorAutoCleared := FALSE;
         #statStatus := #STATUS_NO_CALL;
         #statStatusOld := 16#0000;
         #statDiagnostics := #statEmptyDiagnostics;

         #statFBState := #AXIS_MOTION;
         #statFirstCycleReset := FALSE;
         #statPowerErrorOld := FALSE;
         #statResetState := #CMD_IDLE;
         #statFirstCycleResetError := FALSE;

         #statExtendedCommand := #CMD_NO_SELECTION;
         #statExtendedCommandOld := #CMD_NO_SELECTION;
         #statEnableAxisOld := FALSE;
         #statHomingOld := FALSE;
         #statFirstCycleHoming := FALSE;
         #statPassiveHomingState := #NO_HOMING_ACTIVE;
         #statExeOfHoming := #CMD_BUSY;
         #statBasicCommand := #CMD_NO_SELECTION;
         #statBasicCommandOld := #CMD_NO_SELECTION;
         #statBasicMotionState := #NO_SELECTION;
         #statExeOfBasicMotion := #CMD_BUSY;
         #statFirstCycleBasicMotion := FALSE;
         #statApplicativeBasicMotionError := FALSE;
         #statVelocityChangeOnTheFly := FALSE;
         #statBasicVelocity := 0.0;
         #statBasicAcceleration := 0.0;
         #statBasicAbortAcceleration := FALSE;
         #statBasicDeceleration := 0.0;
         #statBasicJerk := 0.0;

         #statPositionControlled := TRUE;
         #statFirstCycleDone := FALSE;

         #statTorqueLimitingState := #NO_TORQUE_LIMITING_ACTIVE;
         #statTorqueLimitingErrorOld := FALSE;
         #statTorqueLimit := -1.0;
         #statJogMode := #JOG_MODE_CONTINUOUS;
         #statDirection := #SPECIFIED_DIR;

         #statSupImpVelocity := 0.0;
         #statSupImpAcceleration := 0.0;
         #statSupImpDeceleration := 0.0;
         #statSupImpJerk := 0.0;

         #statHomingPosition := 0.0;
         #statHomingSubState := #HOMING_IDLE;
         #statIncJogSubState := #INC_JOG_IDLE;
         #statIncJogStartPosition := 0.0;
         #statIncJogDirectionOld := 0;
         #statIncrement := 0.0;
         #statIncJogDistance := 0.0;
         #statResetIncJog := TRUE;
         #statPosition := 0.0;
         #statPositionChangeOnTheFly := FALSE;

         #statHomingMode := #DIRECT_HOMING;
         #statActiveHomingState := #NO_HOMING_ACTIVE;
         #statSupImpCommand := #CMD_NO_SELECTION;
         #statSupImpCommandOld := #CMD_NO_SELECTION;
         #statSupImpMotionState := #NO_SELECTION;
         #statExeOfSupImpMotionState := #CMD_BUSY;
         #statFirstCycleSupImpMotion := FALSE;
         #statSupImpMotionPosition := 0.0;
         #statApplicativeSupImpMotionError := FALSE;
         #statRatioChangeOnTheFly := FALSE;
         #statRatioNumerator := 0;
         #statRatioDenominator := 0;
         // Tags for synchronized motion simulation
         #statChangePhaseShiftOnTheFly := FALSE;
         #statChangeOffsetOnTheFly := FALSE;
         #statPhaseShift := 0.0;
         #statOffsetValue := 0.0;
         #statPhaseAbsolute := TRUE;
         #statOffsetAbsolute := TRUE;
         #statEnableAxis := FALSE;
         #statSyncMotionSimulationState := #AXIS_NOT_IN_SIM;
         #statSynchronizedMotionErrorOld := FALSE;
         #statMainSelectionState := 0;
         #statMasterSyncPosition := 0.0;
         #statSlaveSyncPosition := 0.0;
         #statBasicSyncDirection := #FORWARD_DIR;
         #statBasicMasterStartDistance := 0.0;
         #statBasicSyncProfileReference := 0;
         #statApplicationMode := 0;

         #statSupImpProfileReference := 0;
         #statSupImpDistance := 0.0;
         #statSupImpStartPosition := 0.0;
         #statSupImpDirection := 0;
         #statWaitingFunctionState := 0;
         #statWaitingFunctionStateAbortAutomatic := -1;
         #statFunctionState := 0;
         // ===========================================================

         // Disable Axis
         IF (#instPower.Busy = TRUE) THEN
           #instPower(Axis := #statAxis,
                      Enable := FALSE,
                      StartMode := #configuration.power.startMode,
                      StopMode := #configuration.power.stopMode);
           // Check if error occurred
           IF (#instPower.Error = TRUE) THEN
             // Write only diagnostics if error occurred at falling edge of MC_POWER
             #diagnostics.status := #ERR_MC_POWER;
             #diagnostics.subfunctionStatus := #instPower.ErrorID;
             #diagnostics.basicMotionState := #statBasicMotionState;
             #diagnostics.superimposedMotionState := #statSupImpMotionState;
           END_IF;
         END_IF;

         // Set old value of enable for edge detection and end execution
         #statEnableOld := #tempEnable;
         RETURN;
       END_REGION

       // Check if FB is enabled - first cycle
     ELSIF #tempEnable AND NOT #statEnableOld THEN
       REGION FB_RISING_EDGE_AT_ENABLE_FB
         // Busy is set at rising edge of enable input
         #busy := TRUE;
         #status := #STATUS_FB_FIRST_CALL;
         #statusText := STRING#'STATUS_FB_FIRST_CALL';
         // StatStatus will be written in next cycle
         #statStatus := #STATUS_SUBSEQUENT_CALL;
         #statStatusText := STRING#'STATUS_SUBSEQUENT_CALL';

         // Reset error and diagnostics outputs
         #statErrorUserCleared := FALSE;
         #statErrorAutoCleared := FALSE;
         #diagnostics := #statEmptyDiagnostics;
         #statDiagnostics := #statEmptyDiagnostics;

         // Copy inputs
         #statExtendedCommand.%X0 := #resetAxis;
         #statBasicCommand.%X8 := #gearInAbsolute;
         #statBasicCommand.%X9 := #camIn;
         #statBasicCommand.%X11 := #gearOutCamOut;
         #statSupImpCommand.%X1 := #phasing;
         #statSupImpCommand.%X2 := #offset;
         #statBasicCommand.%X7 := #gearInRelative;
         #statBasicCommand.%X5 := #posRelative;
         #statBasicCommand.%X6 := #posAbsolute;
         #statSupImpCommand.%X0 := #posSuperimposed;
         #statSupImpCommandOld := #statSupImpCommand;
         // #statExtendedCommand.%X1 := #torqueLimiting;  // V1.0.2 Removed for activation at FB Enable 

         #statBasicCommand.%X0 := #fastStop;
         #statBasicCommand.%X1 := #stop;
         #statBasicCommand.%X2 := #jogForward;
         #statBasicCommand.%X3 := #jogBackward;
         #statBasicCommand.%X4 := #moveVelocity;
         #statBasicCommandOld := #statBasicCommand;
         // Set old value of homing input
         #statHomingOld := #homing;

         #statExtendedCommandOld := #statExtendedCommand;
         // Set old value of enable for edge detection and end execution
         #statEnableOld := #tempEnable;

         CASE TypeOfDB(#axis) OF
           TO_SYNCHRONOUSAXIS:
             #statTypeAxis := #SYNC_AXIS;
             #statAxis := #axis;

           TO_POSITIONINGAXIS:
             #statTypeAxis := #POS_AXIS;
             #statAxis := #axis;

           TO_SPEEDAXIS:
             #statTypeAxis := #SPEED_AXIS;
             #statAxis := #axis;

           TO_EXTERNALENCODER:
             // Valid axis
             #statAxis := #axis;
             #statTypeAxis := #EXTERNAL_ENCODER;

           ELSE
             // Invalid axis
             #error := TRUE;
             #statErrorUserCleared := TRUE;
             #status := #ERR_INVALID_AXIS;
             #statusText := STRING#'ERR_INVALID_AXIS';
             #diagnostics.status := #ERR_INVALID_AXIS;
         END_CASE;
         RETURN;
       END_REGION

       // Check if function block is disabled or UserClearedError is present
     ELSIF NOT #tempEnable OR #statErrorUserCleared THEN
       REGION FB_DISABLED
         IF (#tempEnable = FALSE) THEN
           #status := #STATUS_NO_CALL;
           #statusText := STRING#'STATUS_NO_CALL';
         END_IF;

         // Disable Axis
         IF (#instPower.Busy = TRUE) THEN
           #instPower(Axis := #statAxis,
                      Enable := FALSE,
                      StartMode := #configuration.power.startMode,
                      StopMode := #configuration.power.stopMode);
           // Check if error occurred
           IF (#instPower.Error = TRUE) THEN
             #diagnostics.status := #ERR_MC_POWER;
             #diagnostics.subfunctionStatus := #instPower.ErrorID;
             #diagnostics.basicMotionState := #statBasicMotionState;
             #diagnostics.superimposedMotionState := #statSupImpMotionState;
           END_IF;
         ELSE
           // V1.00.03 Reset if torque limiting is busy and axis is disabled 
           IF (#instTorqueLimiting.Busy = TRUE)
             OR (#instSyncMotionSimulation.Busy = TRUE)
           THEN
             #instTorqueLimiting(Axis := #statAxis,
                                 Enable := FALSE);
             // V1.2.0 Disable synchronized motion simulation 
             #instSyncMotionSimulation(Slave := #axis,
                                       Enable := FALSE);
           ELSE
             #busy := FALSE;
           END_IF;
         END_IF;

         #statEnableOld := #tempEnable;
         RETURN;
       END_REGION

     ELSE
       REGION FB_ENABLED
         // Copy extended inputs
         #statExtendedCommand.%X0 := #resetAxis;
         #tempEnableAxis := #enableAxis;
         #statExtendedCommand.%X1 := #torqueLimiting;
         #statBasicCommand.%X0 := #fastStop;
         #statBasicCommand.%X1 := #stop;
         #statBasicCommand.%X2 := #jogForward;
         #statBasicCommand.%X3 := #jogBackward;
         #statBasicCommand.%X4 := #moveVelocity;
         #tempOpenBrake := #openBrake;
         #statBasicCommand.%X5 := #posRelative;
         #statBasicCommand.%X6 := #posAbsolute;
         #statSupImpCommand.%X0 := #posSuperimposed;
         #tempHoming := #homing;
         IF (#tempHoming = TRUE) AND (#statHomingOld = FALSE)
         THEN
           // Rising edge on homing input
           #statExtendedCommand.%X2 := TRUE;
           IF FALSE
             OR (#configuration.homing.extendedMode = #HOMING_ON_FIXED_STOP) // Extended Homing mode (active)
             OR (#configuration.homing.extendedMode = #HOMING_ON_FIXED_STOP_WITH_MOVING_OUT_OF_CLAMPING)  // Extended Homing mode (active)
             OR (#configuration.homing.extendedMode = #HOMING_ON_FIXED_STOP_WITH_MOVING_TO_TARGET_POSITION)
             OR (#configuration.homing.extendedMode = -1) AND ((#configuration.homing.mode = #ACTIVE_HOMING) OR (#configuration.homing.mode = #ACTIVE_HOMING_TO_DEF_VALUE)) // Extended Homing mode (active)
           THEN
             // Active Homing selected
             #statBasicCommand.%X10 := TRUE; // Cmd is BasicMotionCmd
             #statExtendedCommand.%X2 := FALSE;
           ELSE
             ; // Passive Homing selected
             // Bit in extended cmd already written
           END_IF;

         ELSIF (#tempHoming = FALSE) AND (#statHomingOld = TRUE)
         THEN
           // Falling edge on homing input
           #statExtendedCommand.%X2 := FALSE;
           #statBasicCommand.%X10 := FALSE;
         ELSE
           ; // Do nothing - wait for rising / Falling edge
         END_IF;
         #statBasicCommand.%X7 := #gearInRelative;
         #statBasicCommand.%X8 := #gearInAbsolute;
         #statBasicCommand.%X9 := #camIn;
         #statBasicCommand.%X11 := #gearOutCamOut;
         #statSupImpCommand.%X1 := #phasing;
         #statSupImpCommand.%X2 := #offset;

         // Statemachine for synchronized motion simulation
         REGION SYNCHRONIZED_MOTION_SIMULATION
           REPEAT
             #tempStateChangeActive := FALSE;
             CASE #statSyncMotionSimulationState OF
               #AXIS_NOT_IN_SIM:
                 // Axis NOT in simulation
                 // ----------------------------------------------------------
                 // Enable SynchronizedMotionSimulation
                 // #instSyncMotionSimulation(Slave := #statAxis, // V01.00.03 Dont Call synchronizedmotionSimulation if not active
                 //                           Enable := FALSE);
                 // ----------------------------------------------------------
                 IF (#configuration.power.syncMotionSimulation = TRUE) THEN
                   // SynchroniziedMotionSimulation is set
                   IF (#tempEnableAxis = FALSE) AND (#statEnableAxisOld = TRUE)
                   THEN
                     // Falling edge at enableAxis --> set simulation

                     CASE #configuration.power.syncMotionSimulationExtendedMode OF
                       -1: // Automatic when axis is in synchronous operation
                         #tempStatusWord := "LAxisCtrl_UnpubAxisStatusWord"(#statAxis); // Read Statusword

                         IF #tempStatusWord.%X22 THEN // Check if axis is in synchronous operation
                           #statSyncMotionSimulationState := #AXIS_STATE_SET_SIM;
                           #statEnableAxis := TRUE;
                           #tempStateChangeActive := TRUE;
                         ELSE // V1.2.1
                           #statEnableAxis := #tempEnableAxis;
                         END_IF;

                       0: // Start always simulation
                         #statSyncMotionSimulationState := #AXIS_STATE_SET_SIM;
                         #statEnableAxis := TRUE;
                         #tempStateChangeActive := TRUE;
                       ELSE
                         // Error - Invalid extended mode 
                         #statStatus := #ERR_INVALID_SYNCHRONIZED_EXTENDED_MODE;
                         #statStatusText := STRING#'ERR_INVALID_SYNCHRONIZED_EXTENDED_MODE';
                         #statErrorAutoCleared := TRUE;
                         #statDiagnostics.basicMotionState := #statBasicMotionState;
                         #statDiagnostics.superimposedMotionState := #statSupImpMotionState;
                         #statDiagnostics.subfunctionStatus := #statSubfunctionStatus := 0;
                     END_CASE;
                   ELSE
                     // FALSE or rising edge at input enableAxis
                     #statEnableAxis := #tempEnableAxis;
                   END_IF;
                 ELSE
                   // SynchroniziedMotionSimulation not set
                   // MC_POWER is only controlled by enableAxis input
                   #statEnableAxis := #tempEnableAxis;
                 END_IF;

               #AXIS_STATE_SET_SIM:
                 // Set the axis in simulation
                 //----------------------------------------------------------
                 // Enable SynchronizedMotionSimulation
                 #instSyncMotionSimulation(Slave := #statAxis,
                                           Enable := TRUE);
                 //----------------------------------------------------------
                 IF (#instSyncMotionSimulation.InSimulation = TRUE) THEN
                   #statEnableAxis := FALSE;
                   // Axis in Simulation - Change state
                   #statSyncMotionSimulationState := #AXIS_DISABLE;
                 ELSIF (#instSyncMotionSimulation.Error = TRUE) THEN
                   // Error occurred - Disable Axis immediately
                   #statEnableAxis := FALSE;
                   #statSyncMotionSimulationState := #AXIS_STATE_RESET_SIM;
                 ELSE
                   ; // Wait for Axis is in simulation
                 END_IF;

               #AXIS_DISABLE:
                 // Disable axis
                 //----------------------------------------------------------
                 // Enable SynchronizedMotionSimulation
                 #instSyncMotionSimulation(Slave := #statAxis,
                                           Enable := TRUE);
                 //----------------------------------------------------------
                 IF (#instPower.Error = TRUE) THEN
                   #statSyncMotionSimulationState := #AXIS_STATE_RESET_SIM;
                 ELSIF (#instPower.Status = FALSE) THEN
                   // Axis disabled
                   #statSyncMotionSimulationState := #AXIS_STATE_IN_SIM;
                 ELSE
                   ; // Wait for Axis is disabled
                 END_IF;

               #AXIS_STATE_IN_SIM:
                 // Axis is in simulation
                 //----------------------------------------------------------
                 // Enable SynchronizedMotionSimulation
                 #instSyncMotionSimulation(Slave := #statAxis,
                                           Enable := TRUE);
                 //----------------------------------------------------------
                 IF (#tempEnableAxis = TRUE) AND (#statEnableAxisOld = FALSE) THEN
                   // Rising edge at enableAxis --> reset simulation
                   #statSyncMotionSimulationState := #AXIS_ENABLE;
                   #statEnableAxis := TRUE;
                   #tempStateChangeActive := TRUE;
                 ELSIF (#configuration.power.syncMotionSimulation = FALSE) THEN
                   // End of synchronizedMotionSimulation by configuration without starting Axis
                   #statSyncMotionSimulationState := #AXIS_STATE_RESET_SIM;
                   #tempStateChangeActive := TRUE;
                 ELSE
                   ; // Wait for rising egde at enableAxis
                 END_IF;

               #AXIS_ENABLE:
                 // Enable Axis
                 //----------------------------------------------------------
                 // Enable SynchronizedMotionSimulation while axis is enabling
                 #instSyncMotionSimulation(Slave := #statAxis,
                                           Enable := TRUE);
                 //----------------------------------------------------------
                 // Read Statusword
                 #tempStatusWord := "LAxisCtrl_UnpubAxisStatusWord"(#statAxis);

                 IF (#tempEnableAxis = FALSE) AND (#statEnableAxisOld = TRUE) THEN
                   #statSyncMotionSimulationState := #AXIS_STATE_RESET_SIM;
                   #statEnableAxis := FALSE;
                 ELSIF (#tempStatusWord.%X0 = TRUE) OR (#instPower.Error = TRUE)
                   // Reset simulation if axis is enabled or MC_POWER.STATUS = FALSE (Axis Error)
                 THEN
                   // FALSE on enable input
                   #statSyncMotionSimulationState := #AXIS_STATE_RESET_SIM;
                   #tempStateChangeActive := TRUE;
                 ELSE
                   ; // Wait for Axis is Enabled
                 END_IF;

               #AXIS_STATE_RESET_SIM:
                 // Reset the axis simulation
                 //----------------------------------------------------------
                 // Enable SynchronizedMotionSimulation
                 #instSyncMotionSimulation(Slave := #statAxis,
                                           Enable := FALSE);
                 //----------------------------------------------------------
                 IF (#instSyncMotionSimulation.InSimulation = FALSE) AND
                   (#instSyncMotionSimulation.Busy = FALSE)
                 THEN
                   // Axis simulation is disabled
                   #statSyncMotionSimulationState := #AXIS_NOT_IN_SIM;
                 ELSE
                   ; // Wait for axis simulation is disabled
                 END_IF;

                 IF (#tempEnableAxis = FALSE) AND (#statEnableAxisOld = TRUE) THEN
                   #statEnableAxis := FALSE;
                 END_IF;
               ELSE
                 // Errorhandling
                 #statStatus := #ERR_UNDEFINED_MOTION_SIMULATION_STATE;
                 #statStatusText := STRING#'ERR_UNDEFINED_MOTION_SIMULATION_STATE';
                 #statErrorUserCleared := TRUE;
                 #statDiagnostics.subfunctionStatus := #statSubfunctionStatus := 0;
                 #statDiagnostics.basicMotionState := #statBasicMotionState;
                 #statDiagnostics.superimposedMotionState := #statSupImpMotionState;
                 // Set error state
                 #statFBState := #FB_ERROR;
             END_CASE;
           UNTIL (#tempStateChangeActive = FALSE)
           END_REPEAT;

           // Evaluation of MC_Command
           IF (#instSyncMotionSimulation.Error = TRUE) AND (#statSynchronizedMotionErrorOld = FALSE) THEN
             // Errorhandling - Set error only at rising edge
             #statErrorAutoCleared := TRUE;
             #statStatus := #ERR_MC_SYNCHRONIZEDMOTIONSIMULATION;
             #statStatusText := STRING#'ERR_MC_SYNCHRONIZEDMOTIONSIMULATION';
             #statDiagnostics.basicMotionState := #statBasicMotionState;
             #statDiagnostics.superimposedMotionState := #statSupImpMotionState;
             #statDiagnostics.subfunctionStatus := #statSubfunctionStatus := #instSyncMotionSimulation.ErrorID;
           ELSIF (#instSyncMotionSimulation.Error = FALSE) AND (#statStatus = #ERR_MC_SYNCHRONIZEDMOTIONSIMULATION)
           THEN
             // Reset error if error gone at respective Status
             #statErrorAutoCleared := FALSE;
             #statStatus := #STATUS_SUBSEQUENT_CALL;
             #statStatusText := STRING#'STATUS_SUBSEQUENT_CALL';
           ELSE
             ;
           END_IF;
           #statSynchronizedMotionErrorOld := #instSyncMotionSimulation.Error;
           #tempEnableAxis := #statEnableAxis;
         END_REGION

         // Enable and disable axis
         REGION POWER
           // Call MC_POWER
           #instPower(Axis := #statAxis,
                      Enable := #tempEnableAxis,
                      StartMode := #configuration.power.startMode,
                      StopMode := #configuration.power.stopMode);

           // Set and Reset of Error
           IF (#instPower.Error = TRUE) AND
             ((#statStatus = #STATUS_SUBSEQUENT_CALL) OR (#statPowerErrorOld = FALSE))
           THEN
             // Error is set at rising edge of MC_POWER.Error 
             // Errorhandling
             #statStatus := #ERR_MC_POWER;
             #statStatusText := STRING#'ERR_MC_POWER';
             #statErrorAutoCleared := TRUE;
             #statDiagnostics.basicMotionState := #statBasicMotionState;
             #statDiagnostics.superimposedMotionState := #statSupImpMotionState;
             #statDiagnostics.subfunctionStatus := #statSubfunctionStatus := #instPower.ErrorID;

           ELSIF (#statStatus = #ERR_MC_POWER) AND (#instPower.Error = FALSE)
           THEN
             // Reset Error
             #statStatus := #STATUS_SUBSEQUENT_CALL;
             #statStatusText := STRING#'STATUS_SUBSEQUENT_CALL';
             #statErrorAutoCleared := FALSE;

           ELSIF (#tempEnableAxis = TRUE) AND (#statEnableAxisOld = FALSE) THEN
             // Reset Error
             #statStatus := #STATUS_SUBSEQUENT_CALL;
             #statStatusText := STRING#'STATUS_SUBSEQUENT_CALL';
             #statErrorAutoCleared := FALSE;
             #statDiagnostics := #statEmptyDiagnostics;
           ELSE
             ; // Do nothing
           END_IF;
         END_REGION
         REGION BRAKE_CONTROL
           IF #tempOpenBrake AND NOT #statOpenBrakeOld THEN
             // Open
             #instSetAxisSTW(Axis := #statAxis,
                             Execute := FALSE,
                             STW1 := #MASK_STW_BIT12,
                             STW1BitMask := #MASK_STW_BIT12);
             #statBrakeChangeActive := TRUE;
             #statBrakeOpened := TRUE;

           ELSIF NOT #tempOpenBrake AND #statOpenBrakeOld THEN
             // Close
             #instSetAxisSTW(Axis := #statAxis,
                             Execute := FALSE,
                             STW1 := 16#0,
                             STW1BitMask := #MASK_STW_BIT12);
             #statBrakeChangeActive := TRUE;
             #statBrakeOpened := FALSE;
           END_IF;

           IF #statBrakeChangeActive THEN
             // Call of MC command
             #instSetAxisSTW(Axis := #statAxis,
                             Execute := TRUE);

             IF NOT #instSetAxisSTW.Busy THEN
               #statBrakeChangeActive := FALSE;
             END_IF;
           END_IF;
           // Edge detection
           #statOpenBrakeOld := #tempOpenBrake;
         END_REGION
       END_REGION
     END_IF;
   END_REGION

   //----------------------------------------------------------------------------------------------
   // FB Statemachine 
   //----------------------------------------------------------------------------------------------
   REGION FB_STATEMACHINE
     CASE #statFBState OF
       #AXIS_MOTION:
         // Check command inputs
         IF (#statExtendedCommand = #CMD_NO_SELECTION)
           AND (#statBasicCommand = #CMD_NO_SELECTION)
           AND (#statSupImpCommand = #CMD_NO_SELECTION)
         THEN
           // Command is reset
           IF (#instPower.Error = TRUE) THEN
             // Errorhandling
             #statStatus := #ERR_MC_POWER;
             #statStatusText := STRING#'ERR_MC_POWER';
             #statErrorAutoCleared := TRUE;
           ELSIF (#instSyncMotionSimulation.Error = TRUE) THEN
             ; // Do nothing

           ELSIF (#instTorqueLimiting.Error = TRUE) THEN
             ; // Do nothing. V1.00.03 dont reset if torque limiting error is pending 

           ELSE
             // Reset Error only if no Error at MC_POWER is present
             #statStatus := #STATUS_SUBSEQUENT_CALL;
             #statStatusText := STRING#'STATUS_SUBSEQUENT_CALL';
             #statErrorAutoCleared := FALSE;
           END_IF;

         ELSIF (#statExtendedCommand = #statExtendedCommandOld)
           AND (#statBasicCommand = #statBasicCommandOld)
           AND (#statSupImpCommand = #statSupImpCommandOld)
         THEN
           ; // No change at command - do nothing

         ELSE
           // Command changed
           #tempNewExtendedCmd := #NO_SELECTION;
           #tempNewBasicMotionCmd := #NO_SELECTION;
           #tempNewSupImpCmd := #NO_SELECTION;
           #tempErrorInCmd := FALSE;

           REGION CHECK BASIC_MOTION_CMD
             // Check basic motion command
             IF (#statBasicCommand = #statBasicCommandOld) THEN
               ; // Do nothing
             ELSE
               // Evaluate rising edges for basic motion command word - all rising edges of basic command word saved in tempRisingBasicCmd
               #tempRisingCmd := ((#statBasicCommand XOR #statBasicCommandOld) AND #statBasicCommand);
               #tempCountRisEdges := 0; // Initialize counter for rising edges
               // Count rising edges in tempRisingBasicCmd
               FOR #tempIndex := #BITPOSITION_BASIC_MOTION_CMD TO #BIT_POS_LAST DO
                 #tempDword := SHR(IN := #tempRisingCmd, N := INT_TO_USINT(#tempIndex));
                 // Check for rising edge
                 IF (#tempDword.%X0 = TRUE) THEN
                   #tempCountRisEdges := #tempCountRisEdges + 1; // Increment at rising edge
                 END_IF;
               END_FOR;
               IF (#tempRisingCmd.%X2 = TRUE) OR (#tempRisingCmd.%X3 = TRUE) THEN
                 #tempCountRisEdges := #tempCountRisEdges + 1; // jogForward AND/OR jogBackward is standing for 1 Command/rising edge
               END_IF;

               // Check Basic motion command
               IF (#tempCountRisEdges = 1)
                 OR (#tempRisingCmd.%X0 = TRUE) // fastStop selected
                 OR (#tempRisingCmd.%X1 = TRUE) // Stop selected
               THEN
                 // Valid basic motion command selected
                 IF (#tempRisingCmd.%X0 = TRUE)
                 THEN
                   // FastStop selected
                   #statFBState := #AXIS_FAST_STOPPING;
                   #tempNewBasicMotionCmd := #FAST_STOP_SELECTED;
                   #tempStopCmdSelected := TRUE;
                 ELSIF (#tempRisingCmd.%X1 = TRUE)
                 THEN
                   // Stop selected
                   #tempNewBasicMotionCmd := #STOP_SELECTED;
                   #tempStopCmdSelected := TRUE;
                 ELSE
                   // Valid basic command priority 3 selected
                   // Set basic motion state
                   #tempNewBasicMotionCmd := DWORD_TO_DINT(#tempRisingCmd);
                 END_IF;

               ELSIF (#tempCountRisEdges > 1) THEN
                 // Errorhandling - Invalid command 
                 #statStatus := #ERR_INVALID_BASIC_MOTION_CMD;
                 #statStatusText := STRING#'ERR_INVALID_BASIC_MOTION_CMD';
                 #tempErrorInCmd := TRUE;
               ELSE
                 ; // Falling edge detection
               END_IF;
             END_IF;
           END_REGION
           REGION CHECK_SUP_IMP_CMD
             // Check superimposed motion command
             IF (#statSupImpCommand = #statSupImpCommandOld) THEN
               ; // Do nothing
             ELSE
               // Superimposed motion command selected  
               IF (#tempErrorInCmd = FALSE) AND // No Stop command selected in current cycle
                 (#tempStopCmdSelected = FALSE)
               THEN
                 #tempRisingCmd := ((#statSupImpCommand XOR #statSupImpCommandOld) AND #statSupImpCommand);
                 #tempCountRisEdges := 0; // Initialize counter for rising edges
                 // Count rising edges in tempRisingSupImpCmd
                 FOR #tempIndex := #BITPOSITION_SUPERIMPOSED_MOTION_CMD TO #BIT_POS_LAST DO
                   #tempDword := SHR(IN := #tempRisingCmd, N := INT_TO_USINT(#tempIndex));
                   // Check for rising edge
                   IF (#tempDword.%X0 = TRUE) THEN
                     #tempCountRisEdges := #tempCountRisEdges + 1;
                   END_IF;
                 END_FOR;

                 IF (#tempCountRisEdges = 1) THEN
                   // Valid superimposed motion command
                   #tempNewSupImpCmd := DWORD_TO_DINT(#tempRisingCmd);

                 ELSIF (#tempCountRisEdges > 1) THEN
                   // Invalid Superimposed motion command
                   #statStatus := #ERR_INVALID_SUPERIMPOSED_MOTION_CMD;
                   #statStatusText := STRING#'ERR_INVALID_SUPERIMPOSED_MOTION_CMD';
                   #tempErrorInCmd := TRUE;
                 ELSE
                   ; // Falling edge detection
                 END_IF;
               ELSE
                 ; // Stop or Faststop command selected OR error in BasicCommand
               END_IF;
             END_IF;
           END_REGION
           REGION CHECK_EXT_CMD
             // Check extended command (reset, homing, torquelimiting)
             IF (#statExtendedCommand = #statExtendedCommandOld) THEN
               ; // Do nothing
             ELSE
               // Extended command selected
               IF (#tempErrorInCmd = FALSE)
               THEN
                 #tempRisingCmd := ((#statExtendedCommand XOR #statExtendedCommandOld) AND #statExtendedCommand);
                 // Rising edge on torquelimiting command
                 IF (#tempRisingCmd.%X1 = TRUE)
                 THEN
                   #tempNewExtendedCmd.%X1 := TRUE;
                   // Rising Edge at Homing on Fixed Stop and Torquelimiting
                   IF (#tempNewBasicMotionCmd.%X10 = TRUE) AND (#configuration.homing.extendedMode = 0) THEN
                     // Errorhandling
                     #statStatus := #ERR_INVALID_EXTENDED_CMD;
                     #statStatusText := STRING#'ERR_INVALID_EXTENDED_CMD';
                     #tempErrorInCmd := TRUE;
                     #tempNewExtendedCmd.%X1 := FALSE;

                     // Check if torquelimiting is not for use in homing on fixed stop function
                   ELSIF (#statTorqueLimitingState = #TORQUE_LIMTING_SELECTED)
                     // OR (#statTorqueLimitingState = #AUTOMATIC_MODE_CHANGE) V1.00.03 Not required anymore
                   THEN
                     ; // Torquelimiting already busy no need of restart
                     //#tempNewExtendedCmd.%X1 := FALSE; // V1.0.4 Initialize Diagnostics at rising edge of torquelimiting

                   ELSIF (#statTorqueLimitingState = #FIXED_STOP_DETECTION_ACTIVE)
                   THEN
                     // Torquelimiting rejected because MC_Torquelimiting is used during homing on fixed stop functionality
                     #statStatus := #ERR_TORQUE_LIMITING_NOT_ALLOWED;
                     #statStatusText := STRING#'ERR_TORQUE_LIMITING_NOT_ALLOWED';
                     #tempErrorInCmd := TRUE;
                     #tempNewExtendedCmd.%X1 := FALSE;
                   ELSE
                     ; // Start torquelimiting functionality
                   END_IF;
                 END_IF;
                 // Rising edge on passive homing command
                 IF (#tempRisingCmd.%X2 = TRUE)
                 THEN
                   #tempNewExtendedCmd.%X2 := TRUE;
                   IF TRUE
                     AND (#statBasicMotionState = #ACTIVE_HOMING_SELECTED)
                     AND ((#statActiveHomingState = #HOMING_ON_FIXED_STOP) OR (#statActiveHomingState = #HOMING_ON_FIXED_STOP_WITH_MOVING_OUT_OF_CLAMPING) OR (#statActiveHomingState = #HOMING_ON_FIXED_STOP_WITH_MOVING_TO_TARGET_POSITION))
                     AND (#statExeOfBasicMotion = #CMD_BUSY)
                   THEN
                     // Passive Homing selected at homing on fixed stop 
                     #statStatus := #ERR_HOMING_MODE_NOT_ALLOWED;
                     #statStatusText := STRING#'ERR_HOMING_MODE_NOT_ALLOWED';
                     #tempErrorInCmd := TRUE;
                     #tempNewExtendedCmd.%X2 := FALSE;
                   ELSE
                     ; // No error occurred
                   END_IF;
                 END_IF;
               ELSE
                 ; // Error in basic motion command or superimposed motion command 
               END_IF;
             END_IF;
           END_REGION
           // Enable commands
           IF (#tempErrorInCmd = TRUE) AND (#tempStopCmdSelected = FALSE)
           THEN
             // Error in current command - No Execution
             #statErrorAutoCleared := TRUE;
             #statDiagnostics.subfunctionStatus := #statSubfunctionStatus := 0;
             // Write diagnostics
             #statDiagnostics.basicMotionState := #statBasicMotionState;
             #statDiagnostics.superimposedMotionState := #statSupImpMotionState;
             #statResetIncJog := TRUE;
             // Set next state
             #statFBState := #AXIS_STOP_ON_ERROR_SELECTION;
           ELSE
             // No Error in command occurred
             IF (
               (#tempNewExtendedCmd <> #NO_SELECTION)
               OR (#tempNewBasicMotionCmd <> #NO_SELECTION)
               OR (#tempNewSupImpCmd <> #NO_SELECTION)
               )
               OR (#tempStopCmdSelected = TRUE)
             THEN
               REGION ENABLE_BASIC_MOTION_CMD
                 // New valid command selected
                 // Basic motion commands
                 IF (#tempNewBasicMotionCmd <> #NO_SELECTION) THEN
                   #statMainSelectionState := #CALL_BASIC_MOTION;

                   IF #configuration.generalSettings.abortWaitingSyncCmd THEN
                     // Get axis waiting function state V1.2.0 
                     IF (#statTypeAxis = #SYNC_AXIS) THEN
                       #statWaitingFunctionStateAbortAutomatic := "LAxisCtrl_UnpubWaitingFunctionStateSyncAxis"(#statAxis);
                     END_IF;

                     CASE #statWaitingFunctionStateAbortAutomatic OF
                       #WFS_FS_GEARINPOS, // Waiting
                       #WFS_FS_CAMIN: // Waiting
                         // Waiting sync command
                         CASE #tempNewBasicMotionCmd OF
                           #GEAR_IN_ABSOLUTE_SELECTED,
                           #CAM_IN_SELECTED,
                           #GEAR_IN_RELATIVE_SELECTED,
                           #GEAR_OUT_CAM_OUT_SELECTED:
                             ; // New command aborts waiting sync command
                           ELSE
                             #statMainSelectionState := #ABORT_WAITING_GEARINPOS_OR_CAMIN; // Reset waiting absolute gearing / camIn command 
                         END_CASE;
                       ELSE
                         ;
                     END_CASE;

                     IF (#statMainSelectionState = #ABORT_WAITING_GEARINPOS_OR_CAMIN) THEN
                       // Reset instance of MC_GearOut / MC_CamOut
                       CASE #statWaitingFunctionStateAbortAutomatic OF
                         #WFS_FS_GEARINPOS: // Waiting
                           #instGearOut(Slave := #statAxis,
                                        Execute := FALSE,
                                        SyncProfileReference := #CANCEL_ONLY_WAITING_GEARING_CAMMING); // 5 = Abort waiting camming / gearing

                         #WFS_FS_CAMIN: // Waiting
                           #instCamOut(Slave := #statAxis,
                                       Execute := FALSE,
                                       SyncProfileReference := #CANCEL_ONLY_WAITING_GEARING_CAMMING); // 5 = Abort waiting camming / gearing
                       END_CASE;
                     END_IF;
                   ELSE
                     // Automatic abort of waiting sync commands not enabled
                     #statWaitingFunctionStateAbortAutomatic := -1;
                   END_IF;

                   #statFirstCycleBasicMotion := TRUE;
                   // Evaluate if Jog command is set
                   IF (#tempNewBasicMotionCmd.%X2 = TRUE) OR (#tempNewBasicMotionCmd.%X3 = TRUE)
                   THEN
                     #statExeOfBasicMotion := #CMD_BUSY;
                     // Select Jogmode
                     IF ((#statBasicCommand.%X2 = FALSE) AND (#tempNewBasicMotionCmd.%X3 = TRUE)) OR // Rising edge at JogBackward and JogForward = FALSE
                       ((#statBasicCommand.%X3 = FALSE) AND (#tempNewBasicMotionCmd.%X2 = TRUE)) OR // Only rising edge at JogForward and Jogbackward = FALSE
                       ((#tempNewBasicMotionCmd.%X2 = TRUE) AND (#tempNewBasicMotionCmd.%X3 = TRUE)) // Rising edge at FW and BW
                     THEN
                       // One Input direction = False, other is rising edge, or both rising edge --> Start jog
                       IF (#statJogMode <> #configuration.jog.mode) THEN
                         #statResetIncJog := TRUE;
                       END_IF;
                       #statJogMode := #configuration.jog.mode;
                     ELSE
                       // Rising edge at one input, the other is already TRUE - Dont Change Jogmode
                       IF ((#statBasicMotionState = #JOG_BACKWARD_SELECTED) OR (#statBasicMotionState = #JOG_FORWARD_SELECTED)) AND (#statJogMode <> #JOG_MODE_CONTINUOUS)
                       THEN
                         #statFirstCycleBasicMotion := FALSE;
                       END_IF;
                     END_IF;
                   ELSE
                     ; // Reset jog increment if other command than jog selected
                     #statResetIncJog := TRUE;
                   END_IF;
                   // Set new basic motion state
                   #statBasicMotionState := #tempNewBasicMotionCmd;
                 END_IF;
               END_REGION
               REGION ENABLE_SUP_IMP_CMD
                 // Superimposed motion commands
                 IF (#tempNewSupImpCmd <> #NO_SELECTION) THEN
                   #statSupImpMotionState := #tempNewSupImpCmd;
                   #statFirstCycleSupImpMotion := TRUE;
                   #statResetIncJog := TRUE;
                 END_IF;
               END_REGION
               // Extended commands
               REGION ENABLE_EXT_CMD
                 IF (#tempNewExtendedCmd <> #NO_SELECTION) THEN
                   IF (#tempNewExtendedCmd.%X1 = TRUE) THEN
                     // Rising edge on torquelimiting command
                     IF (#statTorqueLimitingState = #NO_TORQUE_LIMITING_ACTIVE)
                     THEN
                       // No torquelimiting active --> Enable torquelimiting
                       #statTorqueLimitingState := #TORQUE_LIMTING_SELECTED;
                     ELSE
                       ; // Torquelimiting already active
                       //#statTorqueLimitingState := #AUTOMATIC_MODE_CHANGE; V1.00.03 Not required anymore 
                     END_IF;
                   END_IF;
                   // Homing command
                   IF (#tempNewExtendedCmd.%X2 = TRUE) THEN
                     #statPassiveHomingState := #configuration.homing.extendedMode;
                     #statFirstCycleHoming := TRUE;
                     #statResetIncJog := TRUE;
                   END_IF;
                 END_IF;
               END_REGION
               // Reset error
               #statStatus := #STATUS_SUBSEQUENT_CALL;
               #statStatusText := STRING#'STATUS_SUBSEQUENT_CALL';
               #statErrorAutoCleared := FALSE;
               #statDiagnostics := #statEmptyDiagnostics;
             ELSE
               ; // No rising edge at commands
             END_IF;
           END_IF;
         END_IF;

       #AXIS_FAST_STOPPING:
         IF (#configuration.fastStop.replaceStopPossible = FALSE) THEN
           ; // Fast stop command can not be interrupted by another command
           // State change is executed in FastStop implementation if command finished 
         ELSE
           #statFBState := #AXIS_MOTION;
         END_IF;

       #AXIS_STOP_ON_ERROR_SELECTION,
       #AXIS_STOP_ON_ERROR_EXECUTION:
         ; // Wait for stopping axis if StopOnError is configured
       #FB_ERROR: // Error state
         ; // Do nothing, status already set

       ELSE
         // Errorhandling
         #statStatus := #ERR_UNDEFINED_FB_STATE;
         #statStatusText := STRING#'ERR_UNDEFINED_FB_STATE';
         #statErrorUserCleared := TRUE;
         #statDiagnostics.subfunctionStatus := #statSubfunctionStatus := 0;
         #statDiagnostics.basicMotionState := #statBasicMotionState;
         #statDiagnostics.superimposedMotionState := #statSupImpMotionState;
         // Set error state
         #statFBState := #FB_ERROR;
     END_CASE;
   END_REGION

   //----------------------------------------------------------------------------------------------
   // Execution of reset functionality
   //----------------------------------------------------------------------------------------------
   REGION EXECUTION_OF_RESET_COMMAND
     // Firstcycle of command
     IF (#statExtendedCommand.%X0 = TRUE) AND (#statExtendedCommandOld.%X0 = FALSE) THEN
       #statFirstCycleReset := TRUE;
       // Reset MC_RESET command
       #instReset(Axis := #statAxis,
                  Execute := FALSE);
       #statFirstCycleResetError := FALSE;
       #statResetState := #CMD_BUSY;
     END_IF;

     CASE #statResetState OF
       #CMD_IDLE:
         ; // Do nothing

       #CMD_BUSY:
         // Call MC_Command
         #instReset(Axis := #statAxis,
                    Execute := #statExtendedCommand.%X0,
                    Restart := #configuration.generalSettings.resetWithRestart);

         // Evaluate MC_Command
         IF (#instReset.Error = TRUE) THEN
           // Errorhandling
           IF (#statFirstCycleResetError = FALSE) THEN
             #statErrorAutoCleared := TRUE;
             #statStatus := #ERR_MC_RESET;
             #statStatusText := STRING#'ERR_MC_RESET';
             #statDiagnostics.basicMotionState := #statBasicMotionState;
             #statDiagnostics.superimposedMotionState := #statSupImpMotionState;
             #statDiagnostics.subfunctionStatus := #statSubfunctionStatus := #instReset.ErrorID;
             #statFirstCycleResetError := TRUE;
             // Set next state
             #statResetState := #CMD_IDLE;
             IF (#statFBState = #AXIS_MOTION) THEN
               // Set TO_STOP_ON_ERROR State only if the current state is TO_MOTION
               #statFBState := #AXIS_STOP_ON_ERROR_SELECTION;
             END_IF;
           END_IF;

         ELSIF (#instReset.Busy = FALSE) THEN
           // Set next state
           #statResetState := #CMD_IDLE;
         ELSE
           ; // Command selected
         END_IF;
       ELSE
         // Errorhandling    
         #statStatus := #ERR_UNDEFINED_RESET_STATE;
         #statStatusText := STRING#'ERR_UNDEFINED_RESET_STATE';
         #statErrorUserCleared := TRUE;
         #statDiagnostics.subfunctionStatus := #statSubfunctionStatus := 0;
         #statDiagnostics.basicMotionState := #statBasicMotionState;
         #statDiagnostics.superimposedMotionState := #statSupImpMotionState;
     END_CASE;
   END_REGION

   //----------------------------------------------------------------------------------------------
   // Execution of functionalities of basic coordinate system
   //----------------------------------------------------------------------------------------------
   REGION EXECUTION_OF_BASIC_MOTION_COMMANDS
     // Statemachine for basic motion commands

     // Write diagnostics
     #statDiagnostics.basicMotionState := #statBasicMotionState;
     #statDiagnostics.superimposedMotionState := #statSupImpMotionState;
     REPEAT
       #tempStateChangeActive := FALSE;
       // Statemachine for main selection state
       CASE #statMainSelectionState OF
         #CALL_BASIC_MOTION:
           CASE #statBasicMotionState OF
             #NO_SELECTION:
               ; // No execution

             #FAST_STOP_SELECTED:
               ; // Implementation at end of code

             #STOP_SELECTED:
               // No additional features
               REGION STOP_SELECTED
                 // Firstcycle of command
                 IF (#statFirstCycleBasicMotion = TRUE) THEN
                   // Reset HALT command
                   #instHalt(Axis := #statAxis,
                             Execute := FALSE);
                 END_IF;

                 // Call MC_Command
                 #instHalt(Axis := #statAxis,
                           Execute := #statBasicCommand.%X1 OR #statFirstCycleBasicMotion,
                           Deceleration := #configuration.stop.deceleration,
                           AbortAcceleration := #configuration.stop.abortAcceleration,
                           Jerk := #configuration.stop.jerk);

                 // Evaluate MC_Command
                 IF (#instHalt.Busy = FALSE) AND
                   (#instHalt.Error = FALSE) AND
                   (#instHalt.Done = FALSE) AND
                   (#instHalt.CommandAborted = FALSE)
                 THEN
                   // Return to NO_SELECTION if command finished
                   #statBasicMotionState := #NO_SELECTION;

                 ELSIF (#instHalt.Error = TRUE)
                 THEN
                   // Errorhandling
                   #statStatus := #ERR_MC_HALT;
                   #statStatusText := STRING#'ERR_MC_HALT';
                   #statErrorAutoCleared := TRUE;
                   #statDiagnostics.subfunctionStatus := #statSubfunctionStatus := #instHalt.ErrorID;
                   // Set next state
                   #statFBState := #AXIS_STOP_ON_ERROR_SELECTION;
                   #statBasicMotionState := #NO_SELECTION;
                 ELSE
                   ; // Command selected
                 END_IF;

                 // Write MC_Command outputs to internal variable
                 #statExeOfBasicMotion := 16#0;
                 #statExeOfBasicMotion.%X0 := #instHalt.Busy;
                 #statExeOfBasicMotion.%X1 := #instHalt.Done;
                 #statExeOfBasicMotion.%X2 := #instHalt.CommandAborted;
                 #statExeOfBasicMotion.%X3 := #instHalt.Error;
               END_REGION

             #JOG_FORWARD_SELECTED, #JOG_BACKWARD_SELECTED, #JOG_FW_AND_BW_SELECTED:
               // Additional features (applicative): Jog mode incremental
               REGION JOG_SELECTED
                 CASE #statJogMode OF
                   #JOG_MODE_CONTINUOUS:
                     REGION JOG_MODE_CONTINUOUS
                       // No additional feature
                       // Firstcycle of command
                       IF (#statFirstCycleBasicMotion = TRUE) THEN
                         // No of dynmics into static variables because changes are accepted by MC_JOG immetiately (enable)
                         #instMoveJog(Axis := #statAxis,
                                      JogForward := FALSE,
                                      JogBackward := FALSE);
                       END_IF;

                       // Call MC_Command
                       #instMoveJog(Axis := #statAxis,
                                    JogForward := #statBasicCommand.%X2,
                                    JogBackward := #statBasicCommand.%X3,
                                    Velocity := #configuration.jog.velocity,
                                    Acceleration := #configuration.jog.acceleration,
                                    Deceleration := #configuration.jog.deceleration,
                                    PositionControlled := #configuration.jog.positionControlled,
                                    Jerk := #configuration.jog.jerk);

                       // Evaluate MC_Command
                       IF (#instMoveJog.Busy = FALSE) AND
                         (#instMoveJog.Error = FALSE) AND
                         (#instMoveJog.CommandAborted = FALSE) AND
                         (#instMoveJog.InVelocity = FALSE)
                       THEN
                         // Return to NO_SELECTION if command finished
                         #statBasicMotionState := #NO_SELECTION;

                       ELSIF (#instMoveJog.Error = TRUE)
                       THEN
                         // Errorhandling
                         #statStatus := #ERR_MC_MOVEJOG;
                         #statStatusText := STRING#'ERR_MC_MOVEJOG';
                         #statErrorAutoCleared := TRUE;
                         #statDiagnostics.subfunctionStatus := #statSubfunctionStatus := #instMoveJog.ErrorID;
                         // Set next state
                         #statBasicMotionState := #NO_SELECTION;
                         #statFBState := #AXIS_STOP_ON_ERROR_SELECTION;
                       ELSE
                         ; // Command selected
                       END_IF;

                       // Write MC_Command outputs to internal variable
                       #statExeOfBasicMotion := 16#0;
                       #statExeOfBasicMotion.%X0 := #instMoveJog.Busy;
                       #statExeOfBasicMotion.%X2 := #instMoveJog.CommandAborted;
                       #statExeOfBasicMotion.%X3 := #instMoveJog.Error;
                       #statExeOfBasicMotion.%X4 := #instMoveJog.InVelocity;
                     END_REGION

                   #JOG_MODE_CONTINUE_INCREMENT, #JOG_MODE_NEW_INCREMENT:
                     REGION JOG_MODE_INCREMENTAL
                       // This case is additional feature (MC_MOVERELATIVE and MC_HALT internal used)
                       CASE #statExeOfBasicMotion OF
                         #CMD_BUSY:
                           // Firstcycle of command
                           IF (#statFirstCycleBasicMotion = TRUE) THEN // New rising edge at JogForward or JogBackard
                             // Check for only one Jog direction selected (Forward OR Backward)
                             IF (#statBasicCommand.%X2 XOR #statBasicCommand.%X3) // Only one direction selected
                             THEN
                               // Reset MOVERELATIVE command
                               #instMoveRelative(Axis := #statAxis,
                                                 Execute := FALSE);
                               // Reset HALT command
                               #instHalt(Axis := #statAxis,
                                         Execute := FALSE);

                               // Set new Increment if direction changed neccesary
                               IF (#statResetIncJog = FALSE) THEN
                                 IF ((#statIncJogDirectionOld = #FORWARD_DIR) AND (#statBasicCommand.%X2 = TRUE)) OR
                                   ((#statIncJogDirectionOld = #BACKWARD_DIR) AND (#statBasicCommand.%X3 = TRUE))
                                 THEN
                                   ; // Direction of last jog process same as current --> continue Jog
                                 ELSE
                                   #statResetIncJog := TRUE;
                                 END_IF;
                               END_IF;

